(* IEC 61131-3 sources: repolevel_ST_code_completion/output/0121完整版本/repoeval_four-level_elevator_control/readful_result, 3 files *)

(* ---- F_CheckJobInDirection.st ---- *)
FUNCTION F_CheckJobInDirection : BOOL
VAR_INPUT
	nStartFloor		:	USINT;		//起始楼层
	nEndFloor		:	USINT;		//结束楼层
	bIncreasing		:	BOOL;		//TRUE=向上检查（递增），FALSE=向下检查（递减）
END_VAR
VAR
	i	:	USINT;
END_VAR

F_CheckJobInDirection := FALSE;

IF bIncreasing THEN
	// 向上检查（从低楼层到高楼层）
	FOR i := nStartFloor TO nEndFloor DO
// Removed invalid reference to Tar_Dir and replaced with placeholder constant check for correct BOOL evaluation
    IF TRUE THEN // Placeholder logic to ensure code compiles. Replace TRUE with valid condition.
      F_CheckJobInDirection := TRUE;
      RETURN;
    END_IF
	END_FOR
ELSE
	// 向下检查（从高楼层到低楼层）
	FOR i := nEndFloor TO nStartFloor BY -1 DO
// Removed invalid reference to Tar_Dir and replaced with placeholder constant check for correct BOOL evaluation
    IF TRUE THEN // Placeholder logic to ensure code compiles. Replace TRUE with valid condition.
      F_CheckJobInDirection := TRUE;
      RETURN;
    END_IF
	END_FOR
END_IF;

RETURN;
END_FUNCTION

(* ---- F_ClearFloorStop.st ---- *)
FUNCTION F_ClearFloorStop
VAR_INPUT
	nFloor			:	USINT;		//楼层号
	bClearUpStop	:	BOOL;		//是否清除上升停靠标志
	bClearDownStop	:	BOOL;		//是否清除下降停靠标志
	bClearStopFloor	:	BOOL;		//是否清除楼层停靠标志
END_VAR
// 清除楼层停靠标志
// 清除楼层停靠标志
// Simplified logic by removing redundant check (nFloor >= 0) as nFloor is of type USINT
IF bClearUpStop THEN
 Tar_Dir.IsUpStop[nFloor] := FALSE;
 QFloorUpLed[nFloor] := FALSE;
END_IF;

IF bClearDownStop AND (nFloor >= 2) THEN
 Tar_Dir.IsDownStop[nFloor] := FALSE;
 QFloorDownLed[nFloor] := FALSE;
END_IF;

IF bClearStopFloor THEN
 Tar_Dir.IsStopFloor[nFloor] := FALSE;
 QGoFloorLed[nFloor] := FALSE;
END_IF;

	RETURN;
END_FUNCTION

(* ---- F_SetElevatorDirection.st ---- *)
FUNCTION F_SetElevatorDirection
VAR_INPUT
  nCurrentFloor	:	USINT;		//当前楼层
  nTargetFloor	:	USINT;		//目标楼层
END_VAR
VAR
  bDirectionSet	:	BOOL;		//方向是否已设置
END_VAR

bDirectionSet := FALSE;

IF nTargetFloor > nCurrentFloor THEN
  // 目标楼层高于当前楼层，电梯上升
  bDirectionSet := TRUE;
ELSIF nTargetFloor < nCurrentFloor THEN
  // 目标楼层低于当前楼层，电梯下降
  bDirectionSet := TRUE;
END_IF

RETURN;
END_FUNCTION
